FUNCTION_BLOCK VISU
VAR_INPUT
END_VAR
VAR_OUTPUT
END_VAR
VAR
END_VAR

END_FUNCTION_BLOCK

(* stored: Version 1.1.0.1, ProductVersion 3.1.4024.16
   POU VISU: Id {8c79f4c1-9909-4056-b77f-242d9e2e78d9}, SpecialFunc None *)
